(*

.. <legal notes>

legal notes
=================
| SPDX-FileCopyrightText: © 2025 Oleksandr Tiutyk <trofimich@gmail.com>
| SPDX-License-Identifier: LGPL-3.0-only
| For details check: LGPL-3.0-only_

.. _LGPL-3.0-only: https://www.gnu.org/licenses/lgpl-3.0.en.html

.. </legal notes>

*)

TYPE AUTOMATION_RUNNER_DIAGNOSTICS :
STRUCT
	HandleEnabledStateError : AUTOMATION_RUNNER_ERROR_LOG;
	HandleSimulationModeStateError : AUTOMATION_RUNNER_ERROR_LOG;
	
	InitializationError : AUTOMATION_RUNNER_ERROR_LOG;
	
	CriticalRunningOrStopingError : AUTOMATION_RUNNER_ERROR_LOG;
	
	LastRuningNonCriticalError : AUTOMATION_RUNNER_ERROR_LOG;
	LastStopingNonCriticalError : AUTOMATION_RUNNER_ERROR_LOG;
	
	HandleFaultError : AUTOMATION_RUNNER_ERROR_LOG;	
END_STRUCT
END_TYPE

(* stored: Version 1.1.0.1
   DUT AUTOMATION_RUNNER_DIAGNOSTICS: Id {abe4ac9d-925d-4d89-96b8-639221428dee} *)
